Staubli VAL3: writeDET.pgx

program writeDET()
  local bool l_bResult
  local num l_nError
  local string l_sValue
begin
  // Update variables of the conveyor library
  resize(sCaption,1,pg:nNumOfTxtBox)
  call pg:getCaption(sCaption)
  // Buffersize
  call pg:getFieldValue(sCaption[0],l_sValue,l_nError)
  toNum(l_sValue,det:nMaxNumOfObject,l_bResult)
end
